// TIA Portal V20 export
TYPE "LWONIK_typeWinderMode"
// stored: Access Published
   STRUCT
      unwinderLeftUse : Bool;
      unwinderRightUse : Bool;
      rewinderLeftUse : Bool;
      rewinderRightUse : Bool;
   END_STRUCT;
END_TYPE
